# EPICS substitutions: db/ecmcIPOS8020_AUX.substitutions
file ecmcIPOSXXXX_AUX.template
{
	pattern {CURRESLO}
		{0.001221}
}
